(* PLC project Unnamed, Unknown Unnamed 1 *)
(* stored: creationDateTime 2026-02-24T10:48:54, modificationDateTime 2026-02-24T10:55:06 *)

PROGRAM program0
  VAR
    X : INT := 5;
    Y : INT := 2;
    Q : INT;
  END_VAR

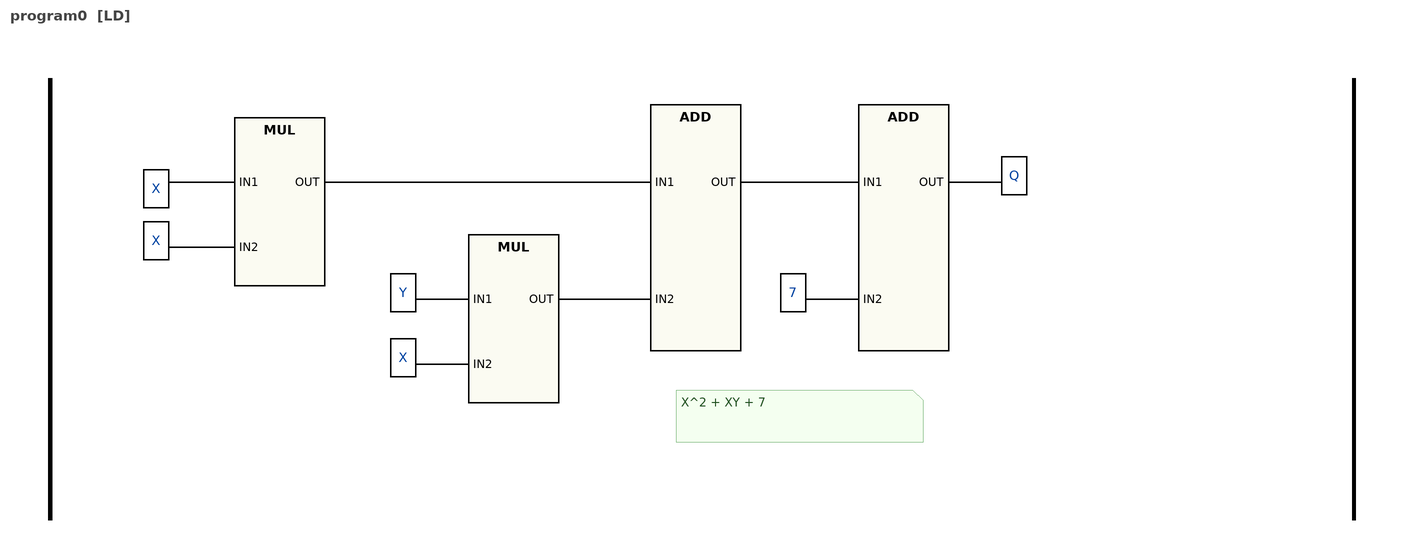
(* LD diagram, written out as Structured Text *)
Q := X * X + Y * X + 7;
(* X^2 + XY + 7 *)
END_PROGRAM

CONFIGURATION Config0
  RESOURCE Res0 ON PLC
    TASK task0(INTERVAL := T#20ms, PRIORITY := 0);
    PROGRAM instance0 WITH task0 : program0;
  END_RESOURCE
END_CONFIGURATION
